{attribute 'linkalways'}
{attribute 'no_explicit_call' := 'This FB is a CLASS and must be accessed using methods or properties'}
{attribute 'enable_dynamic_creation'}
FUNCTION_BLOCK Node_F_VN_TransformCoordinatesPlanar_Point EXTENDS VisionNode
VAR
    aSrcPoint : _TcVnPoint2_LREAL;
    aDestPoint : _TcVnPoint2_LREAL;
    aTransformationMatrix : _TcVnMatrix3x3_LREAL;
    hrPrev : _HRESULT(S_OK);
    hresult : _HRESULT(S_OK);
END_VAR

METHOD PUBLIC Clone : I_Node
VAR
    pNode : POINTER TO Node_F_VN_TransformCoordinatesPlanar_Point;
END_VAR
pNode := __NEW(Node_F_VN_TransformCoordinatesPlanar_Point);
Clone := pNode^;
END_METHOD

METHOD FB_init : BOOL
VAR_INPUT
    bInitRetains : BOOL;
    bInCopyCode : BOOL;
END_VAR
AddInput('aSrcPoint', aSrcPoint);
AddInput('aTransformationMatrix', aTransformationMatrix);
AddInput('hrPrev', hrPrev);
AddOutput('aDestPoint', aDestPoint);
AddOutput('hresult', hresult);
END_METHOD

METHOD PROTECTED OnExecute
hresult.Value := F_VN_TransformCoordinatesPlanar_Point(
    aSrcPoint := aSrcPoint.Value,
    aDestPoint := aDestPoint.Value,
    aTransformationMatrix := aTransformationMatrix.Value,
    hrPrev := hrPrev.Value);
END_METHOD

METHOD PUBLIC PreExecutionCheck
VAR_INPUT
    Check : I_PreExecutionChecks;
END_VAR
Check.IsTrue(aTransformationMatrix.Value[2, 2] <> 0.0, 'aTransformationMatrix must be a valid transformation matrix (connect a planar calibration result)');
END_METHOD

END_FUNCTION_BLOCK

(* stored: Version 1.1.0.1, ProductVersion 3.1.4026.19
   POU Node_F_VN_TransformCoordinatesPlanar_Point: Id {5b9fd172-dc91-4cf0-b90e-34adef22196f}, SpecialFunc None
   Folder Constructor: Id {5eb3e0c9-dba7-42ba-a52b-7fedf6c09a79}
   Method Clone: Id {c66362aa-bca4-492e-b22a-705d35f98692}
   Method FB_init: Id {1ab62d46-e4a5-4aeb-b3bc-bfcab95ac423}
   Method OnExecute: Id {d7cda93f-e293-4e1d-babd-25773c69999a}
   Method PreExecutionCheck: Id {07593510-fbe5-47a4-8f18-ab616ee46e87} *)
